{attribute 'OPC.UA.DA.StructuredType' := '1'}
FUNCTION_BLOCK FB_PumpDOL_Onga413_RND EXTENDS FB_BaseDevice IMPLEMENTS I_Device, I_PumpVSD

VAR
	bFirstRun: BOOL := TRUE;
	{attribute 'OPC.UA.DA' := '1'} 
	bInContactor AT %I*: BOOL := FALSE;
	{attribute 'OPC.UA.DA' := '1'} 
	bOutContactor AT %Q*: BOOL := FALSE;

	
	fbTON_OnTimer: TON := (PT := tTimeOn, IN := FALSE);
	tTimeOn: TIME := T#15S;
	
	//MB:  REFERENCE TO FB_ModbusMaster;
	{attribute 'OPC.UA.DA' := '1'}
	nFrequencySetPoint: REAL := 0;
	{attribute 'OPC.UA.DA' := '1'}
	nFrequencyActual: REAL := 0;
	
	{attribute 'OPC.UA.DA' := '0'} 
	eSMState: (WAIT, STARTING, RUNNING, STOPPING, STOPPED);
	
	tDebounce: TIME := T#5S;
	fbTON_Debounce: TON := (PT := tDebounce, IN := FALSE);
	
END_VAR

IF bFirstRun THEN
	bFirstRun := FALSE;

END_IF

fbTON_Debounce();
fbTONstartTime(PT := tTimeOn);
fbTON_OnTimer(PT := tTimeOn);
fbTONstopTime();



IF GVL.bAutoUpdateDeviceState THEN
	eState := eStateTarget;	
END_IF




IF eMode = E_DeviceMode.MANUAL THEN
	bEnable := TRUE;
END_IF

IF bEnable AND (eStateTarget = E_DeviceState.RUNNING) AND eSMState <> RUNNING THEN
		eSMState := STARTING;
		fbTON_Debounce(IN := TRUE);
		fbTON_OnTimer(IN := TRUE);
		
END_IF

IF (bEnable = FALSE OR eStateTarget = E_DeviceState.IDLE) AND eSMState <> WAIT THEN
		eSMState := STOPPING;
		fbTON_Debounce(IN := FALSE);
		fbTON_OnTimer(IN := FALSE);
END_IF


(*

CASE eSMState OF
	
	WAIT:
		//Wait for method call to change ESMState
		fbTON_OnTimer(IN := FALSE);
		
	STARTING: 
	
		IF fbTON_Debounce.Q THEN
			eState := E_DeviceState.STARTING;
			fbTON_OnTimer(IN := TRUE);
			bOutContactor := TRUE;
		
			IF fbTONstartTime.Q THEN
				eSMState := WAIT;
				raiseAlarm(Priority := E_AlarmPriority.High, Label := 'Failed to Start', Enabled := TRUE, DeviceAlarmID := 1);
			END_IF
			
			IF TRUE THEN
				eSMState := RUNNING;
				eState := E_DeviceState.RUNNING;
			END_IF
			fbTON_Debounce(IN := FALSE);
		END_IF

		
	RUNNING:
		IF bOutContactor <> TRUE THEN
			raiseAlarm(Priority := E_AlarmPriority.High, Label := 'Power Lost', Enabled := TRUE, DeviceAlarmID := 2);
			eState := E_DeviceState.IDLE;
			eSMState := WAIT;
		END_IF
		
		// Add pump / motor control here - look at built in Twincat libraries 
		// Add relevant VSD signals to check
		

	STOPPING:
		eState := E_DeviceState.STOPPING;
		bOutContactor := FALSE;
		eSMState := STOPPED;

		

	STOPPED:
		eState := E_DeviceState.IDLE;
		fbTON_Debounce(IN := TRUE);
		eSMState := WAIT;
		
		
END_CASE

*)

CASE eSMState OF
	
	WAIT:
		//Wait for method call to change ESMState
		
	STARTING: 
		IF fbTON_Debounce.Q THEN
			eState := E_DeviceState.STARTING;
			bOutContactor := TRUE;
			fbTON_Debounce.IN := FALSE;
			eSMState := RUNNING;
		END_IF

		
	RUNNING:
		eState := E_DeviceState.RUNNING;
		IF bOutContactor <> TRUE THEN
			raiseAlarm(Priority := E_AlarmPriority.High, Label := 'Power Lost', Enabled := TRUE, DeviceAlarmID := 1);
			eSMState := STOPPING;
		END_IF
			
	STOPPING:
		fbTON_Debounce.IN := TRUE;
		fbTON_OnTimer(IN := FALSE);
		bOutContactor := TRUE;
		eState := E_DeviceState.STOPPING;
		bOutContactor := FALSE;
		eSMState := STOPPED;

	STOPPED:
		eState := E_DeviceState.IDLE;
		eSMState := WAIT;
		fbTON_Debounce.IN := TRUE;
		
END_CASE

{warning 'add method implementation '}
METHOD disable : BOOL
bEnable := FALSE;
END_METHOD

{warning 'add method implementation '}
METHOD enable : BOOL
bEnable := TRUE;
END_METHOD

{warning 'add method implementation '}
METHOD FB_init : BOOL
VAR_INPUT
	(* if TRUE, the retain variables are initialized (warm start / cold start)*)
	bInitRetains	: BOOL;
	(* if TRUE, the instance afterwards gets moved into the copy code (online change)*)
	bInCopyCode	: BOOL;
	PumpID	: STRING(80);
	PumpDescr	: STRING(255);
END_VAR
sID := PumpID;
sDescr := PumpDescr;
END_METHOD

{warning 'add method implementation '}
METHOD getFrequency : REAL
END_METHOD

METHOD setModbusMaster : BOOL
METHOD setModbusMaster : BOOL
VAR_INPUT
	//ModbusMaster: REFERENCE TO FB_ModbusMaster;
END_VAR
//MB := ModbusMaster;
END_METHOD

METHOD setOff : BOOL
VAR_INPUT
END_VAR
END_METHOD

METHOD setOn : BOOL
VAR_INPUT
END_VAR
END_METHOD

{warning 'add method implementation '}
METHOD setReference : BOOL
VAR_INPUT
	RefSetPoint	: REAL;
END_VAR
END_METHOD

METHOD startTimer : BOOL
VAR_INPUT
END_VAR
startTimer := fbTON_OnTimer.Q;
END_METHOD

END_FUNCTION_BLOCK

(* stored: Version 1.1.0.1, ProductVersion 3.1.4024.12
   POU FB_PumpDOL_Onga413_RND: Id {4b5eeba4-a037-4613-9994-e90d3fc96810}, SpecialFunc None
   Method disable: Id {3d3c54a2-89a2-40aa-a306-832de325e18f}
   Method enable: Id {4932c99d-c1c6-4be0-bb48-f110cf873cdc}
   Method FB_init: Id {fd98e5ce-e559-4759-bc79-9bc4526aeeed}
   Method getFrequency: Id {ce11ccdd-6f8b-4a4b-842e-589c9a033792}
   Method setModbusMaster: Id {10695257-924e-4032-a7d2-d94b686bd899}
   Method setOff: Id {833dfaa6-eee6-4104-ac2d-b7d8d0dbdfd7}
   Method setOn: Id {88075d38-edf7-46fe-bea7-194a7f200d47}
   Method setReference: Id {f7724c37-3f96-404d-89e2-812e72ef800c}
   Method startTimer: Id {58f0f73a-01ed-4c12-ab65-50b709290395} *)
